Universal Robots PolyScope program: HeatPTemUreduce10.urp

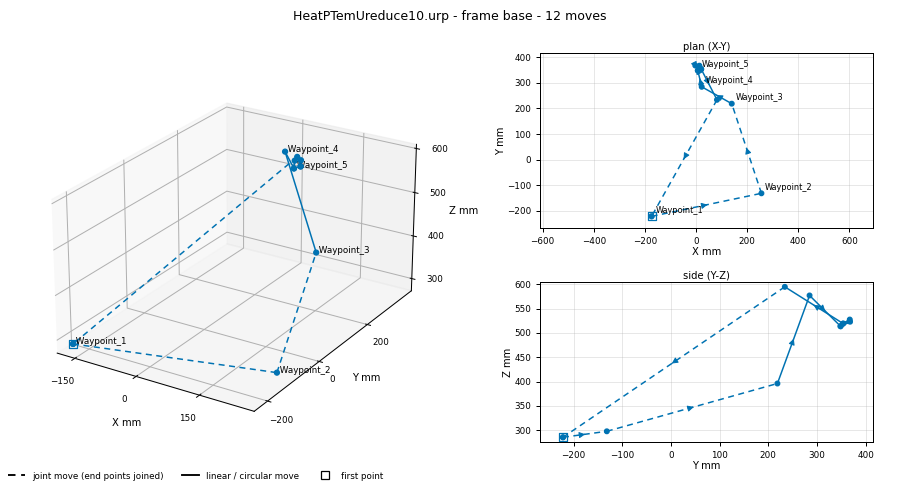
[picture p0: tool path of HeatPTemUreduce10.urp in frame base, 12 of 12 moves have a stored position in this frame; points joined in program order, loops and branches not executed]
Program TDHeatPTemUreduce10 (installation=default directory=/programs/usbdisk_0/UR_URPs createdIn=5.11.0.108249 lastSavedIn=5.11.0.108249 robotSerialNumber=20215590035)
Calibrated DH parameters: a=[0.00016, -0.349388, -0.392209, -0.000059, 0.000026, 0]; d=[0.162575, -215.770964, 216.209801, -0.305241, 0.099656, 0.099253]; alpha=[1.570834, -0.001122, 0.007322, 1.56929, -1.570073, 0]; deltaTheta=[0, 0.606034, 5.685341, -0.008192, 0.000001, 0]
Robot Program (runOnlyOnce=true)
  MoveJ speed 60 deg/s, acceleration 80 deg/s^2 (useActiveTCP=true) feature=Base
    Waypoint Waypoint_1: TCP in base x=-173.939 y=-221.905 z=285.6 mm, rx=-2.1904 ry=-2.2352 rz=0.015 rad; joints [-99.419, -57.385, -139.029, -73.574, 89.583, 79.477] deg; TCP offset x=0 y=0 z=26 mm, rx=0 ry=0 rz=0 rad
  MoveJ speed 60 deg/s, acceleration 80 deg/s^2 (useActiveTCP=true) feature=Base
    Waypoint Waypoint_2: TCP in base x=255.607 y=-131.807 z=297.919 mm, rx=-0.0229 ry=3.1151 rz=-0.0378 rad; joints [1.04, -57.382, -137.549, -73.627, 89.053, 90.235] deg
  MoveJ speed 60 deg/s, acceleration 80 deg/s^2 (useActiveTCP=true) feature=Base
    Waypoint Waypoint_3: TCP in base x=139.565 y=218.746 z=396.126 mm, rx=-2.1977 ry=2.2399 rz=-0.0498 rad; joints [89.241, -50.957, -124.715, -95.52, 89.056, 90.235] deg
  URCap Gripper Activate (Robotiq_Grippers, Robotiq Inc.) dataModel(ResetAndActivateKey=false)
  URCap Gripper (Robotiq_Grippers, Robotiq Inc.) dataModel(position=0.0, force=99.6078431372549, speed=99.6078431372549, positionInDouble=0.0, forceInDouble=99.6078431372549, speedInDouble=99.6078431372549, slaveIds=[9], blocking=true)
  MoveP speed 250 mm/s, acceleration 1200 mm/s^2 (blendRadius=0.025 useActiveTCP=true) feature=Base
    Waypoint Waypoint_4: TCP in base x=22.115 y=284.761 z=577.036 mm, rx=-1.2884 ry=1.2268 rz=1.1411 rad; joints [137.343, -43.027, -132.051, -11.67, 43.033, 92.524] deg
  MoveL speed 250 mm/s, acceleration 1200 mm/s^2 (useActiveTCP=true) feature=Base
    Waypoint Waypoint_5: TCP in base x=6.838 y=348.415 z=513.773 mm, rx=-1.292 ry=1.2795 rz=1.0343 rad; joints [126.817, -59.243, -135.03, 3.891, 49.347, 92.313] deg
  MoveL speed 250 mm/s, acceleration 1200 mm/s^2 (useActiveTCP=true) feature=Base
    Waypoint Waypoint_6: TCP in base x=-2.916 y=367.941 z=523.156 mm, rx=-1.2893 ry=1.3646 rz=0.9906 rad; joints [126.613, -61.633, -131.104, -2.766, 47.649, 97.367] deg
  MoveL speed 250 mm/s, acceleration 1200 mm/s^2 (useActiveTCP=true) feature=Base
    Waypoint Waypoint_5: TCP in base x=6.838 y=348.415 z=513.773 mm, rx=-1.292 ry=1.2795 rz=1.0343 rad; joints [126.817, -59.243, -135.03, 3.891, 49.347, 92.313] deg
  MoveL speed 250 mm/s, acceleration 1200 mm/s^2 (useActiveTCP=true) feature=Base
    Waypoint Waypoint_7: TCP in base x=20.153 y=353.825 z=519.301 mm, rx=-1.2941 ry=1.3286 rz=1.0268 rad; joints [122.707, -59.629, -133.311, 0.669, 52.959, 94.358] deg
  Loop Counting (count=10) loopVariable(name=Loop_1)
    MoveL speed 250 mm/s, acceleration 1200 mm/s^2 (useActiveTCP=true) feature=Base
      Waypoint Waypoint_8: TCP in base x=13.093 y=367.397 z=527.544 mm, rx=-1.3297 ry=1.3406 rz=0.9655 rad; joints [122.705, -61.196, -130.377, -3.98, 52.186, 94.336] deg
    MoveL speed 250 mm/s, acceleration 1200 mm/s^2 (useActiveTCP=true) feature=Base
      Waypoint Waypoint_7: TCP in base x=20.153 y=353.825 z=519.301 mm, rx=-1.2941 ry=1.3286 rz=1.0268 rad; joints [122.707, -59.629, -133.311, 0.669, 52.959, 94.358] deg
  MoveL speed 250 mm/s, acceleration 1200 mm/s^2 (useActiveTCP=true) feature=Base
    Waypoint Waypoint_9: TCP in base x=81.811 y=233.934 z=594.753 mm, rx=-1.4214 ry=1.3335 rz=1.1037 rad; joints [121.814, -34.693, -127.276, -33.232, 61.608, 96.375] deg
  MoveJ speed 60 deg/s, acceleration 80 deg/s^2 (useActiveTCP=true) feature=Base
    Waypoint Waypoint_1: TCP in base x=-173.939 y=-221.905 z=285.6 mm, rx=-2.1904 ry=-2.2352 rz=0.015 rad; joints [-99.419, -57.385, -139.029, -73.574, 89.583, 79.477] deg
  URCap Gripper (Robotiq_Grippers, Robotiq Inc.) dataModel(position=100.0, force=99.6078431372549, speed=99.6078431372549, positionInDouble=100.0, forceInDouble=99.6078431372549, speedInDouble=99.6078431372549, slaveIds=[9], blocking=true)
